{region '#Template'}
	{attribute 'Version' := '1.2.1.0'}
	{attribute 'Tags' := '"LCID": "1031", "Text": "Universal, Sensor, AI"'}
	{attribute 'Tags' := '"LCID": "1033", "Text": "Universal, Sensor, AI"'}
	{attribute 'Using' := '"Type": "Template", "URI": "EC_AMEV"'}
	{attribute 'Using' := '"Type": "Template", "URI": "BA2_Param"'}
	{attribute 'Description' := '"LCID": "1031", "Text": "Kombination 4x AI ohne IO"'}
	{attribute 'Description' := '"LCID": "1033", "Text": "Combination 4x AI without IO"'}
{endregion}
FUNCTION_BLOCK FB_BA_MeasuredValueCardinal EXTENDS FB_BA_View
VAR_INPUT
	fVal_N					: REAL;
	fVal_S					: REAL;
	fVal_E					: REAL;
	fVal_W					: REAL;
END_VAR
VAR_INPUT CONSTANT
	MV_N					: FB_BA_AI;		
	MV_S					: FB_BA_AI;	
	MV_E					: FB_BA_AI;		
	MV_W					: FB_BA_AI;			
END_VAR
VAR_OUTPUT
	fPresentValueN			: REAL;
	fPresentValueS			: REAL;
	fPresentValueE			: REAL;
	fPresentValueW			: REAL;
END_VAR
VAR
END_VAR

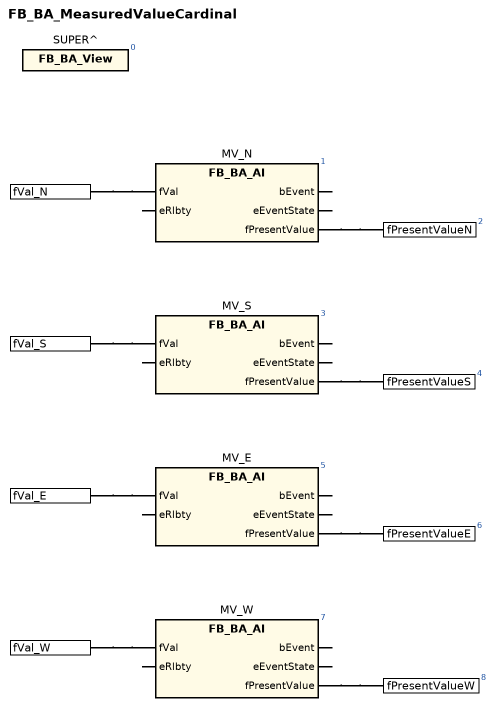
SUPER^(); // FB_BA_View
MV_N(fVal := fVal_N); // FB_BA_AI
fPresentValueN := MV_N.fPresentValue;
MV_S(fVal := fVal_S); // FB_BA_AI
fPresentValueS := MV_S.fPresentValue;
MV_E(fVal := fVal_E); // FB_BA_AI
fPresentValueE := MV_E.fPresentValue;
MV_W(fVal := fVal_W); // FB_BA_AI
fPresentValueW := MV_W.fPresentValue;

METHOD FB_init : BOOL
VAR_INPUT
	bInitRetains : BOOL; // if TRUE, the retain variables are initialized (warm start / cold start)
	bInCopyCode : BOOL;  // if TRUE, the instance afterwards gets moved into the copy code (online change)
END_VAR
MV_N.iParent						:= THIS^;		
MV_N.iLabel 						:= LblUniFieldDevice.SensorAnalog_MV_N;
MV_N.sObjectName					:= '{Idx=01}';
MV_N.sDeviceType					:= '';
MV_N.bEnOutOfService				:= FALSE;
MV_N.eUnit							:= E_BA_Unit.eTemperature_DegreesCelsius;
MV_N.fCOVIncrement					:= BA2_Param.fDefCOVIncrement;
MV_N.nEventClassID					:= EC_ID.NC30;
MV_N.stTimeDelay.nToNormal			:= BA2_Param.nDefTimeDelay_ToNormal;
MV_N.stTimeDelay.nToAbnormal		:= BA2_Param.nDefTimeDelay_ToAbnormal;
MV_N.stHighLimit.bEnable			:= FALSE;
MV_N.stHighLimit.fValue				:= 0.0;		
MV_N.stLowLimit.bEnable				:= FALSE;
MV_N.stLowLimit.fValue				:= 0.0;
MV_N.fLimitDeadband 				:= BA2_Param.fDefLimitDeadband;
MV_N.bAcknowledgeRm					:= FALSE;	
MV_N.aEventTransitionText[1]		:= txtEvent_Exceeded;
MV_N.aEventTransitionText[2]		:= txtEvent_Disturb;
MV_N.aEventTransitionText[3]		:= txtEvent_Normal;
MV_N.bEventDetectionEnable			:= FALSE;
MV_N.aEventEnable[1]				:= TRUE;			//	to_offnormal
MV_N.aEventEnable[2]				:= TRUE;			//	to_fault
MV_N.aEventEnable[3]				:= TRUE;			//	to_normal
MV_N.eEnPlantLock					:= E_BA_LockPriority.eNoLock;			

MV_S.iParent						:= THIS^;		
MV_S.iLabel 						:= LblUniFieldDevice.SensorAnalog_MV_S;
MV_S.sObjectName					:= '{Idx=02}';
MV_S.sDeviceType					:= '';
MV_S.bEnOutOfService				:= FALSE;
MV_S.eUnit							:= E_BA_Unit.eTemperature_DegreesCelsius;
MV_S.fCOVIncrement					:= BA2_Param.fDefCOVIncrement;
MV_S.nEventClassID					:= EC_ID.NC30;
MV_S.stTimeDelay.nToNormal			:= BA2_Param.nDefTimeDelay_ToNormal;
MV_S.stTimeDelay.nToAbnormal		:= BA2_Param.nDefTimeDelay_ToAbnormal;
MV_S.stHighLimit.bEnable			:= FALSE;
MV_S.stHighLimit.fValue				:= 0.0;		
MV_S.stLowLimit.bEnable				:= FALSE;
MV_S.stLowLimit.fValue				:= 0.0;
MV_S.fLimitDeadband 				:= BA2_Param.fDefLimitDeadband;
MV_S.bAcknowledgeRm					:= FALSE;	
MV_S.aEventTransitionText[1]		:= txtEvent_Exceeded;
MV_S.aEventTransitionText[2]		:= txtEvent_Disturb;
MV_S.aEventTransitionText[3]		:= txtEvent_Normal;
MV_S.bEventDetectionEnable			:= FALSE;
MV_S.aEventEnable[1]				:= TRUE;			//	to_offnormal
MV_S.aEventEnable[2]				:= TRUE;			//	to_fault
MV_S.aEventEnable[3]				:= TRUE;			//	to_normal
MV_S.eEnPlantLock					:= E_BA_LockPriority.eNoLock;

MV_E.iParent						:= THIS^;		
MV_E.iLabel 						:= LblUniFieldDevice.SensorAnalog_MV_E;
MV_E.sObjectName					:= '{Idx=03}';
MV_E.sDeviceType					:= '';
MV_E.bEnOutOfService				:= FALSE;
MV_E.eUnit							:= E_BA_Unit.eTemperature_DegreesCelsius;
MV_E.fCOVIncrement					:= BA2_Param.fDefCOVIncrement;
MV_E.nEventClassID					:= EC_ID.NC30;
MV_E.stTimeDelay.nToNormal			:= BA2_Param.nDefTimeDelay_ToNormal;
MV_E.stTimeDelay.nToAbnormal		:= BA2_Param.nDefTimeDelay_ToAbnormal;
MV_E.stHighLimit.bEnable			:= FALSE;
MV_E.stHighLimit.fValue				:= 0.0;		
MV_E.stLowLimit.bEnable				:= FALSE;
MV_E.stLowLimit.fValue				:= 0.0;
MV_E.fLimitDeadband 				:= BA2_Param.fDefLimitDeadband;
MV_E.bAcknowledgeRm					:= FALSE;	
MV_E.aEventTransitionText[1]		:= txtEvent_Exceeded;
MV_E.aEventTransitionText[2]		:= txtEvent_Disturb;
MV_E.aEventTransitionText[3]		:= txtEvent_Normal;
MV_E.bEventDetectionEnable			:= FALSE;
MV_E.aEventEnable[1]				:= TRUE;			//	to_offnormal
MV_E.aEventEnable[2]				:= TRUE;			//	to_fault
MV_E.aEventEnable[3]				:= TRUE;			//	to_normal
MV_E.eEnPlantLock					:= E_BA_LockPriority.eNoLock;

MV_W.iParent						:= THIS^;		
MV_W.iLabel 						:= LblUniFieldDevice.SensorAnalog_MV_W;
MV_W.sObjectName					:= '{Idx=04}';
MV_W.sDeviceType					:= '';
MV_W.bEnOutOfService				:= FALSE;
MV_W.eUnit							:= E_BA_Unit.eTemperature_DegreesCelsius;
MV_W.fCOVIncrement					:= BA2_Param.fDefCOVIncrement;
MV_W.nEventClassID					:= EC_ID.NC30;
MV_W.stTimeDelay.nToNormal			:= BA2_Param.nDefTimeDelay_ToNormal;
MV_W.stTimeDelay.nToAbnormal		:= BA2_Param.nDefTimeDelay_ToAbnormal;
MV_W.stHighLimit.bEnable			:= FALSE;
MV_W.stHighLimit.fValue				:= 0.0;		
MV_W.stLowLimit.bEnable				:= FALSE;
MV_W.stLowLimit.fValue				:= 0.0;
MV_W.fLimitDeadband 				:= BA2_Param.fDefLimitDeadband;
MV_W.bAcknowledgeRm					:= FALSE;	
MV_W.aEventTransitionText[1]		:= txtEvent_Exceeded;
MV_W.aEventTransitionText[2]		:= txtEvent_Disturb;
MV_W.aEventTransitionText[3]		:= txtEvent_Normal;
MV_W.bEventDetectionEnable			:= FALSE;
MV_W.aEventEnable[1]				:= TRUE;			//	to_offnormal
MV_W.aEventEnable[2]				:= TRUE;			//	to_fault
MV_W.aEventEnable[3]				:= TRUE;			//	to_normal
MV_W.eEnPlantLock					:= E_BA_LockPriority.eNoLock;
END_METHOD

END_FUNCTION_BLOCK

(* stored: Version 1.1.0.1, ProductVersion 3.1.4024.9
   POU FB_BA_MeasuredValueCardinal: Id {d0dda666-5e23-44c9-a243-fc08620492da}, SpecialFunc None
   Method FB_init: Id {8651e786-db88-4c5e-8048-b3fc9befdaac} *)
